FUNCTION_BLOCK APPEND_STRING_2
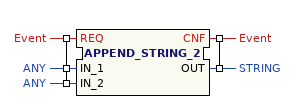
  EVENT_INPUT
    REQ WITH IN_1, IN_2;
  END_EVENT
  EVENT_OUTPUT
    CNF WITH OUT;
  END_EVENT
  VAR_INPUT
    IN_1 : ANY;
    IN_2 : ANY;
  END_VAR
  VAR_OUTPUT
    OUT : STRING;
  END_VAR
END_FUNCTION_BLOCK
